FUNCTION_BLOCK TcoComponentTest EXTENDS TcoCore._internals_TcoContext
VAR
	_callMyPlcInstance	:	BOOL := FALSE;
	_component : _TcoComponent(THIS^);
	_runPLCinstanceOnce : BOOL := FALSE;
	_runPLCinstanceCyclicaly : BOOL := FALSE;
	_restore : BOOL;
	_cycleCount : INT;
	_restoreCycleCount : INT;
	_init: BOOL;
END_VAR

IF _callMyPlcInstance THEN
	IF NOT _init THEN
		ContextOpen();	
		ContextClose();	
		_init := THIS^._rtc.IsValid;
	END_IF
	
	IF _restore THEN
		ContextOpen();	
		THIS^._component.Restore();	
		_restoreCycleCount := _restoreCycleCount + 1;
		_restore := FALSE;
		ContextClose();	
		RETURN;
	END_IF
	
	IF _runPLCinstanceOnce AND NOT _runPLCinstanceCyclicaly THEN
		ContextOpen();	
		THIS^.PLCinstanceRun();
		_cycleCount := _cycleCount + 1;
		_runPLCinstanceOnce := FALSE;
		ContextClose();	
	END_IF
	
	IF _runPLCinstanceCyclicaly AND NOT _runPLCinstanceOnce THEN
		ContextOpen();	
		THIS^.PLCinstanceRun();
		_cycleCount := _cycleCount + 1;
		ContextClose();	
	END_IF
END_IF;

{attribute 'TcRpcEnable'}
METHOD INTERNAL ContextClose
SUPER^._Close();
END_METHOD

{attribute 'TcRpcEnable'}
METHOD INTERNAL ContextOpen
SUPER^._Open();
END_METHOD

{attribute 'TcRpcEnable'}
METHOD INTERNAL IsService : BOOL
IsService := THIS^._component.IsService;
END_METHOD

METHOD PROTECTED  Main
END_METHOD

{attribute 'TcRpcEnable'}
METHOD INTERNAL PLCinstanceRun
THIS^._component();
END_METHOD

METHOD PROTECTED Restore
THIS^._component.Restore();
END_METHOD

{attribute 'TcRpcEnable'}
METHOD INTERNAL Service
THIS^._component.Service();
END_METHOD

{attribute 'TcRpcEnable'}
METHOD INTERNAL TriggerRestore
THIS^.Restore();
END_METHOD

END_FUNCTION_BLOCK

(* stored: Version 1.1.0.1
   POU TcoComponentTest: Id {b7fdd050-d5b9-04ff-0c52-b3ea7a75470a}, SpecialFunc None
   Method ContextClose: Id {4b2d831f-b02d-0dc7-1aba-0c0212f05248}
   Method ContextOpen: Id {a232ffc8-ce87-0a52-3e0f-8790c172b4db}
   Method IsService: Id {492ba7c1-2102-0be5-16e2-886c69f0ee52}
   Method Main: Id {c9c7735e-2c49-0853-1698-e16c59099e7f}
   Method PLCinstanceRun: Id {a455bb82-c564-00ec-161f-5a8a7b4faa57}
   Method Restore: Id {5d28ce32-be6d-072a-02e9-9e3a46400612}
   Method Service: Id {12499dae-6b36-0f57-3ded-b8b2964f6cd4}
   Method TriggerRestore: Id {b586ab69-4eb0-05bd-2907-c9b7d8f8b9e2} *)
